// TIA Portal V20 export
TYPE "LER_typeBrakeTestEmStatus"
// stored: Access Published
   STRUCT
      axisEnabled { ExternalWritable := 'False'} : Array[0..49] of Bool;
      busy { ExternalWritable := 'False'} : Array[0..49] of Bool;
      complete { ExternalWritable := 'False'} : Array[0..49] of Bool;
   END_STRUCT;
END_TYPE
